{attribute 'no_explicit_call' := 'do not call this FB directly'}{attribute 'enable_dynamic_creation'}
FUNCTION_BLOCK InputPort_ANY EXTENDS Disposable IMPLEMENTS I_InputPort
VAR
	_name : T_MAXSTRING;
	_permittedDataTypes : T_MAXSTRING;
	_connectedTo : I_OutputPort;
	internalBuffer : POINTER TO BYTE;
	internalBufferSize : UDINT;
	eventEmitter : EventEmitter;
END_VAR

METHOD PUBLIC Accept
VAR_INPUT
	Visitor : I_InputPortVisitor;
END_VAR
Visitor.VisitInputPort(this^);
END_METHOD

METHOD PRIVATE CheckSourceDataTypeIsAllowed : BOOL
VAR_INPUT
	Source : I_OutputPort;
END_VAR
VAR
	searchString : T_MAXSTRING;
	leftString : T_MAXSTRING;
	rightString : T_MAXSTRING;
END_VAR
IF PermittedDataTypes = '' THEN 
	CheckSourceDataTypeIsAllowed := TRUE;
	RETURN;;
END_IF

IF PermittedDataTypes = Source.DataType THEN 	
	CheckSourceDataTypeIsAllowed := TRUE;
	RETURN;
END_IF

searchString := PermittedDataTypes;

WHILE findAndSplitChar(sSeparatorChar := ',', pSrcString := ADR(searchString), pLeftString := ADR(leftString), nLeftSize := SIZEOF(leftString), pRightString := ADR(rightString), nRightSize := SIZEOF(rightString), bSearchFromRight := FALSE) DO 

	IF leftString = Source.DataType OR rightString = Source.DataType THEN 	
		CheckSourceDataTypeIsAllowed := TRUE;
		RETURN;
	END_IF
	
	searchString := rightString;

END_WHILE
END_METHOD

METHOD PUBLIC ConnectTo
VAR_INPUT
	OutputPort : I_OutputPort;
END_VAR
IF NOT CheckSourceDataTypeIsAllowed(OutputPort) THEN
	RETURN;
END_IF

OutputPort.OnEvent('OnOutputPortChanged', THIS^);
_connectedTo := OutputPort;
END_METHOD

METHOD PRIVATE CopyInternalBufferToDestination
VAR_INPUT
	DestinationAddress : PVOID;
END_VAR
memcpy(DestinationAddress,internalBuffer,internalBufferSize);
END_METHOD

METHOD PRIVATE CopySourceToInternalBuffer
VAR_INPUT
	SourceAddress : PVOID;
END_VAR
memcpy(internalBuffer,SourceAddress,internalBufferSize);
END_METHOD

PROPERTY PUBLIC DataSize : UDINT
GET
IF internalBuffer = 0 THEN
	RETURN;
END_IF

DataSize := internalBufferSize;
END_GET
END_PROPERTY

PROPERTY PUBLIC DataType : T_MAXSTRING
GET
IF NOT IsConnected THEN 
	RETURN;
END_IF

DataType := _connectedTo.DataType;
END_GET
END_PROPERTY

METHOD PRIVATE DeleteInternalBuffer
IF internalBuffer <> 0 THEN
	__DELETE(internalBuffer);
END_IF
END_METHOD

METHOD PUBLIC Disconnect
IF _connectedTo = 0 THEN
	RETURN;
END_IF

_connectedTo.OffEvent('OnOutputPortChanged', THIS^);
_connectedTo := 0;
END_METHOD

METHOD PRIVATE EmitOnInputPortChangeEvent
VAR_INPUT
	PortChanged : I_InputPort;
END_VAR
VAR
	pInputPortChangeEvent : POINTER TO InputPortChangedEvent;
END_VAR
pInputPortChangeEvent := __NEW(InputPortChangedEvent(TargetInputPort := PortChanged));
eventEmitter.Emit('OnInputPortChanged',pInputPortChangeEvent^);
pInputPortChangeEvent^.Dispose();
END_METHOD

METHOD FB_exit : BOOL
VAR_INPUT
	bInCopyCode : BOOL; // if TRUE, the exit method is called for exiting an instance that is copied afterwards (online change).
END_VAR
IF bInCopyCode THEN
	RETURN;
END_IF

DeleteInternalBuffer();
END_METHOD

METHOD FB_init : BOOL
VAR_INPUT
	bInitRetains : BOOL; // if TRUE, the retain variables are initialized (warm start / cold start)
	bInCopyCode : BOOL;  // if TRUE, the instance afterwards gets moved into the copy code (online change)
	Name : T_MAXSTRING;
	PermittedDataTypes : T_MAXSTRING;
	Parent : I_HaveInputPorts;
END_VAR
_name := Name;
_permittedDataTypes := PermittedDataTypes;

IF Parent = 0 THEN
	RETURN;
END_IF

Parent.AddInputPort(THIS^);
END_METHOD

METHOD PUBLIC Get
VAR_INPUT
	Value : ANY;
END_VAR
GetTo(Value.pValue, DINT_TO_UDINT(Value.diSize));
END_METHOD

METHOD PUBLIC GetTo
VAR_INPUT
	Destination : PVOID;
	DestinationSize : UDINT;
END_VAR
IF NOT IsInternalBufferSameSizeAs(DestinationSize) THEN
	RETURN;
END_IF

CopyInternalBufferToDestination(Destination);
END_METHOD

METHOD PUBLIC HandleEvent
VAR_INPUT
	Event : I_Event;
END_VAR
VAR
	outputPortChangedEvent : I_OutputPortChangedEvent;
END_VAR
IF __QUERYINTERFACE(Event, outputPortChangedEvent) THEN
	HandleOutputPortChangedEvent(outputPortChangedEvent.TargetOutputPort);
END_IF
END_METHOD

METHOD PUBLIC HandleOutputPortChangedEvent
VAR_INPUT
	Source : I_OutputPort;
END_VAR
DeleteInternalBuffer();

IF NOT CheckSourceDataTypeIsAllowed(Source) THEN
	RETURN;
END_IF

MakeInternalBufferOfSize(Source.DataSize);
Source.GetTo(internalBuffer,internalBufferSize);

EmitOnInputPortChangeEvent(THIS^);
END_METHOD

PROPERTY HasData : BOOL
GET
IF NOT IsConnected THEN 
	RETURN;
END_IF

HasData := _connectedTo.HasData;
END_GET
END_PROPERTY

PROPERTY PUBLIC IsConnected : BOOL
GET
IsConnected := _connectedTo <> 0;
END_GET
END_PROPERTY

METHOD PRIVATE IsInternalBufferSameSizeAs : BOOL
VAR_INPUT
	Size : UDINT;
END_VAR
IF internalBuffer = 0 THEN
	RETURN;
END_IF

IF internalBufferSize <> Size THEN
	RETURN;
END_IF

IsInternalBufferSameSizeAs := TRUE;
END_METHOD

METHOD PRIVATE MakeInternalBufferOfSize
VAR_INPUT
	Size : UDINT;
END_VAR
internalBufferSize := Size;
internalBuffer := __NEW(BYTE, internalBufferSize);
END_METHOD

PROPERTY PUBLIC Name : T_MAXSTRING
GET
Name := _name;
END_GET
END_PROPERTY

METHOD PUBLIC OffEvent
VAR_INPUT
	EventName : T_MaxString;
	EventHandler : I_EventHandler;
END_VAR
eventEmitter.OffEvent(EventName, EventHandler);
END_METHOD

METHOD PUBLIC OnceEvent
VAR_INPUT
	EventName : T_MaxString;
	EventHandler : I_EventHandler;
END_VAR
eventEmitter.OnceEvent(EventName, EventHandler);
END_METHOD

METHOD PUBLIC OnEvent
VAR_INPUT
	EventName : T_MaxString;
	EventHandler : I_EventHandler;
END_VAR
eventEmitter.OnEvent(EventName, EventHandler);
END_METHOD

PROPERTY PUBLIC PermittedDataTypes : T_MAXSTRING
GET
PermittedDataTypes := _permittedDataTypes;
END_GET
END_PROPERTY

METHOD PUBLIC Set
VAR_INPUT
	Value : ANY;
END_VAR
SetFrom(Value.pValue, DINT_TO_UDINT(Value.diSize));
END_METHOD

METHOD PUBLIC SetFrom
VAR_INPUT
	SourceAddress : PVOID;
	SourceSize : UDINT;
END_VAR
DeleteInternalBuffer();
MakeInternalBufferOfSize(SourceSize);
CopySourceToInternalBuffer(SourceAddress);
EmitOnInputPortChangeEvent(this^);
END_METHOD

END_FUNCTION_BLOCK

(* stored: Version 1.1.0.1, ProductVersion 3.1.4024.12
   POU InputPort_ANY: Id {8a76cd64-8399-006f-0213-1bb5b2341bca}, SpecialFunc None
   Folder Constructor: Id {c02273f4-e8fc-0d09-3c19-79f73fa57a1b}
   Folder Destructor: Id {ba2ea5f2-36a9-0932-19c7-fcbc4ffe5fb3}
   Folder Private: Id {1f1fa75f-3537-0229-2498-8638fd4c140f}
   Method Accept: Id {1625d170-79e2-014d-2c2b-8ace06c47aa1}
   Method CheckSourceDataTypeIsAllowed: Id {cf78df18-286c-090f-1ebf-1b4924ebafa2}
   Method ConnectTo: Id {cf2a22c3-c119-0919-3767-3381d146e55b}
   Method CopyInternalBufferToDestination: Id {d780866f-a8a9-0d8b-14ce-acf2a3dc97e8}
   Method CopySourceToInternalBuffer: Id {ecd1f6d6-3198-0f94-3d6b-8138401f05d7}
   Property DataSize: Id {3d8fffe6-ccba-0ff2-0252-789287dd2651}
   Get Get: Id {9b02a0ef-8be9-0d14-1f38-bd3f727f753d}
   Property DataType: Id {f697d0c9-35bd-003b-2eed-d1db3a1aaa7d}
   Get Get: Id {9027c130-d714-0b66-2e0c-fed40c3b84cf}
   Method DeleteInternalBuffer: Id {099abdf9-5e01-0ce5-1920-94b1d39942de}
   Method Disconnect: Id {2d2d97fa-faba-033e-23df-3b334614454b}
   Method EmitOnInputPortChangeEvent: Id {c9ad38c0-e6a0-080d-0291-a5f6bdd88e5d}
   Method FB_exit: Id {5bbffd23-4d4b-08bd-2200-a37d8613dfbf}
   Method FB_init: Id {85cb6971-3869-03dd-0362-0b78635177f7}
   Method Get: Id {f813caa3-f9f5-0763-25b7-95603e18c9c7}
   Method GetTo: Id {6cdee704-352c-0268-1a5b-c9cf7fee8290}
   Method HandleEvent: Id {a301251b-128e-042e-2c82-4ee90daa8459}
   Method HandleOutputPortChangedEvent: Id {9bdbd293-4e3d-0e2f-0079-1e62c2ac0372}
   Property HasData: Id {028c08e7-27ab-0342-09cc-9dbc235ca19c}
   Get Get: Id {18f5535a-a48c-01cf-11dc-2957e3d7d564}
   Property IsConnected: Id {0eeca197-140f-0917-0914-20aa772b83ae}
   Get Get: Id {7caf9676-d732-0ed2-375f-00350fceb01e}
   Method IsInternalBufferSameSizeAs: Id {4b5eee94-77e1-0a27-1a14-11203e2f0f97}
   Method MakeInternalBufferOfSize: Id {1e9e66b3-85ba-06d2-3b40-d013d15273d1}
   Property Name: Id {bed621d8-5fb5-029d-2ec1-72a1805573da}
   Get Get: Id {81e0229a-69c1-0712-0a6c-c9c3a3d10c8f}
   Method OffEvent: Id {8831601f-10ed-0308-0255-7aeb488c0bb1}
   Method OnceEvent: Id {02751623-dd18-0013-0361-602d9e5793b3}
   Method OnEvent: Id {6400660c-9990-0d44-03fa-8885dfec75cf}
   Property PermittedDataTypes: Id {756bbe97-8ed1-003d-213d-e72af1469808}
   Get Get: Id {cd1c0acd-4bfd-0274-050d-5fc5fc240ae1}
   Method Set: Id {11bb708a-c074-063b-3b6f-6f91adf498fb}
   Method SetFrom: Id {a0fdb2f8-cbff-0fe3-1955-a0d3bea340b0} *)
